// TIA Portal V21 export
VAR_GLOBAL   // PLC tag table "DI"
   "EMG SWITCH" AT %I0.0 : Bool;
   "RESET PB" AT %I0.1 : Bool;
   "VACUUM PUMP TRIP" AT %I0.2 : Bool;
   "DOOR1 OPEN LMT" AT %I0.3 : Bool;
   "DOOR1 CLOSE LMT" AT %I0.4 : Bool;
   "DOOR2 OPEN LMT" AT %I0.5 : Bool;
   "DOOR2 CLOSE LMT" AT %I0.6 : Bool;
   "DOOR2 CLOSE PB" AT %I0.7 : Bool;
   "DOOR2 OPEN PB" AT %I1.0 : Bool;
   "DOOR1 CLOSE PB" AT %I1.1 : Bool;
   "DOOR1 OPEN PB" AT %I1.2 : Bool;
   "AIR PREESURE SWS" AT %I1.3 : Bool;
   "plant steam low" AT %I1.4 : Bool;
   "pure steam low" AT %I1.5 : Bool;
   "cooling wtr low" AT %I2.0 : Bool;
   SPP AT %I2.1 : Bool;
   "DOOR1 CURTAIN SENSOR" AT %I2.2 : Bool;
   "DOOR2 CURTAIN SENSOR" AT %I2.3 : Bool;
   "BOILER WATER LEVEL OK" AT %I2.4 : Bool;
   "DRUM VFD TRIP" AT %I10.2 : Bool;
   "CRC PUMP TRIP" AT %I10.4 : Bool;
END_VAR
